TYPE ty_Motor_Outputs :
STRUCT
    // Physical Output (Выход на реле/контактор)
    b_Activate_Contactor             : BOOL;
    
    // Status Flags
    b_Motor_IsRunning                : BOOL;
    b_MotorError                     : BOOL;
END_STRUCT
END_TYPE

(* stored: Version 1.1.0.1
   DUT ty_Motor_Outputs: Id {c0a5b483-ebdf-4182-9b7b-b0e1d73e8f09} *)
